FUNCTION_BLOCK PAMHopperscale EXTENDS PAProcessModule
VAR_INPUT
END_VAR
VAR_OUTPUT
END_VAR
VAR
	_PAPointMatIn1 : PAPoint(THIS^);
	_PAPointMatOut1 : PAPoint(THIS^);
END_VAR

METHOD FB_init : BOOL
VAR_INPUT
	bInitRetains : BOOL; // if TRUE, the retain variables are initialized (warm start / cold start)
	bInCopyCode : BOOL;  // if TRUE, the instance afterwards gets moved into the copy code (online change)
	parent : IACComponent;
END_VAR
AddPoint(_PAPointMatIn1);
AddPoint(_PAPointMatOut1);
END_METHOD

PROPERTY PUBLIC PAPointMatIn1 : IACPoint
GET
PAPointMatIn1 := _PAPointMatIn1;
END_GET
END_PROPERTY

PROPERTY PUBLIC PAPointMatOut1 : IACPoint
GET
PAPointMatOut1 := _PAPointMatOut1;
END_GET
END_PROPERTY

END_FUNCTION_BLOCK

(* stored: Version 1.1.0.1, ProductVersion 3.1.4020.12
   POU PAMHopperscale: Id {e641740c-06ba-466d-a5e6-22d0379ea510}, SpecialFunc None
   Method FB_init: Id {a93a8873-ca21-4dcb-8d67-c54595bfe395}
   Property PAPointMatIn1: Id {b129d6bf-1558-4cba-909a-6de1937430db}
   Get Get: Id {251488a2-4af2-49a3-92d5-9467ac666da7}
   Property PAPointMatOut1: Id {bb66304f-bcb1-4c90-a930-a8753194ae4f}
   Get Get: Id {7637d192-0cee-4495-8020-9b4110b6a476} *)
